# EPICS alarm handler configuration: apps/alh/ecal.alhConfig
#===============================================================================
# ECAL Alarm Config
#===============================================================================

GROUP NULL ECAL

#=======================================
# Subsystems
#=======================================

INCLUDE ECAL /usr/clas12/hps/prod/apps/alh/hv.alhConfig
INCLUDE ECAL /usr/clas12/hps/prod/apps/alh/tempSens.alhConfig
